ABB RobotStudio station: Project1_3.rspag

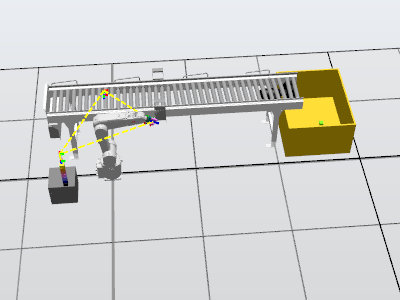
--- station ---
Station Project1 (saved by RobotStudio 23.3.10550.0)
Controller Controller1
  mechanical unit ROB_1: IRB1200_5_90_STD_03, 6 joints, base frame (0, 0, 0) mm
Layout (positions relative to the parent item):
  - My_Gripper_Mech [mechanism] at (461.39, 0, 883.1) mm, rotated rx 180 ry 60 rz 180 deg; joint values [0, 0] (rad or m)
      TCP My_Gripper_Mech_1 at (0, 0, 70) mm
      links: L1, L2, L3
  - LineSensor [smart component, from Components\LineSensor.rslib] at (522.01, 0, 848.1) mm, rotated rx 180 ry 60 rz 180 deg
      properties: Start=[0 0 0]; End=[0 0 0.1]; Length=0.1; Radius=0; Tag=(none); SensedPart=(none); SensedPoint=[0 0 0]
    - _sensorPart_ [part, from Components\LineSensor.rslib]
  - Attacher [smart component, from Components\Attacher.rslib]
      properties: Parent=IRB1200_5_90_STD_03; Flange=0; Child=(none); Mount=false; Offset=[0 0 0]; Orientation=[0 0 0]
  - Detacher [smart component, from Components\Detacher.rslib]
      properties: Child=(none); KeepPosition=true
  - PoseMover [smart component, from Components\PoseMover.rslib]
      properties: Mechanism=My_Gripper_Mech; Pose=1; Duration=0
  - PoseMover_2 [smart component, from Components\PoseMover.rslib]
      properties: Mechanism=My_Gripper_Mech; Pose=2; Duration=0
  - puelko [part] at (-800, -100, 0) mm, size 800 x 1000 x 500 mm
  - klocek8 [part] at (-525, -400, 300) mm, size 50 x 50 x 50 mm
  - klocek7 [part] at (-525, -400, 350) mm, size 50 x 50 x 50 mm
  - klocek6 [part] at (-525, -400, 400) mm, size 50 x 50 x 50 mm
  - IRB1200_5_90_STD_03 [mechanism, from %ABB.RobotStudio.Models.IRB1200%\IRB1200_5_90_STD_03.rslib] at (0, 0, 0) mm; joint values [0, -0.1239, 0.0383, 0, 0.6093, 0] (rad or m)
  - 400_guide [part, from %ABB.RobotStudio.Models.Conveyors%\Conveyor Guide 400.rslib] at (-700, 401, -100) mm
  - klocek3 [part] at (-525, -400, 550) mm, size 50 x 50 x 50 mm
  - klocek5 [part] at (-525, -400, 450) mm, size 50 x 50 x 50 mm
  - klocek4 [part] at (-525, -400, 500) mm, size 50 x 50 x 50 mm
  - Part_1 [part] at (0, -100, 0) mm, size 300 x 300 x 200 mm
  - klocek2 [part] at (-525, -400, 600) mm, size 50 x 50 x 50 mm
  - klocek1 [part] at (2609.57, 581.28, -0.23) mm, rotated rx -89.6 ry -89.83 rz -4.57 deg, size 50 x 50 x 50 mm
  - Part_3 [part] at (0, 0, 0) mm, size 300 x 300 x 100 mm
Attachment: LineSensor is attached to My_Gripper_Mech / L1
Attachment: My_Gripper_Mech is attached to IRB1200_5_90_STD_03 / Link6
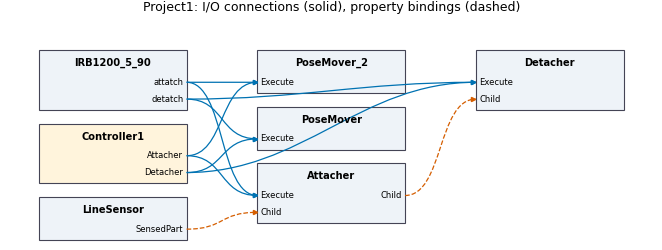
Station logic (signal -> signal, property => property):
  IRB1200_5_90.attatch -> Attacher.Execute
  IRB1200_5_90.detatch -> Detacher.Execute
  IRB1200_5_90.attatch -> PoseMover_2.Execute
  IRB1200_5_90.detatch -> PoseMover.Execute
  Controller1.Attacher -> Attacher.Execute
  Controller1.Detacher -> Detacher.Execute
  Controller1.Attacher -> PoseMover_2.Execute
  Controller1.Detacher -> PoseMover.Execute
  Attacher.Child => Detacher.Child
  LineSensor.SensedPart => Attacher.Child

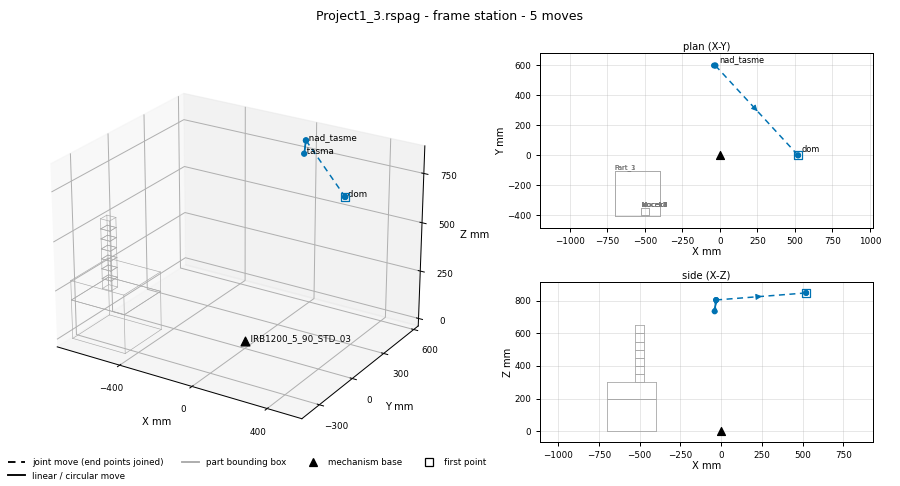
[picture p0: tool path of Project1_3.rspag in frame station, 5 of 8 moves have a stored position in this frame; points joined in program order, loops and branches not executed]
--- Controller Data/Controller1/RAPID/TASK1/PROGMOD/CalibData.mod ---
MODULE CalibData
    PERS tooldata My_Gripper_Mech_1:=[TRUE,[[0,0,70],[1,0,0,0]],[1,[1,1,1],[1,0,0,0],0,0,0]];
    TASK PERS wobjdata Workobject_1:=[FALSE,TRUE,"",[[0,0,0],[1,0,0,0]],[[0,0,0],[1,0,0,0]]];
    PERS tooldata My_Gripper_Mech_1_2:=[TRUE,[[0,0,70],[1,0,0,0]],[1,[1,1,1],[1,0,0,0],0,0,0]];
ENDMODULE

--- Controller Data/Controller1/RAPID/TASK1/PROGMOD/Module1.mod ---
MODULE Module1
    CONST robtarget dom:=[[522.01408311,0,848.1],[0.5,0,0.866025404,0],[0,0,0,0],[9E+09,9E+09,9E+09,9E+09,9E+09,9E+09]];
    CONST robtarget nad_klocek:=[[-500,-375,810],[0,0.707106781,0.707106781,0],[-2,0,-1,0],[9E+09,9E+09,9E+09,9E+09,9E+09,9E+09]];
    CONST robtarget klocek:=[[-500,-375,700],[0,0.707106781,0.707106781,0],[-2,0,-1,0],[9E+09,9E+09,9E+09,9E+09,9E+09,9E+09]];
    CONST robtarget nad_tasme:=[[-30.156,599.226,805],[0,1,0,0],[0,0,-2,0],[9E+09,9E+09,9E+09,9E+09,9E+09,9E+09]];
    CONST robtarget tasma:=[[-39.156,599.226,735],[0,1,0,0],[0,0,-2,0],[9E+09,9E+09,9E+09,9E+09,9E+09,9E+09]];
    VAR robtarget nad_klocekvar;
    VAR robtarget klocekvar;
    PROC Path_10()
        FOR z FROM 0 TO 0 DO
            nad_klocekvar:=Offs(nad_klocek,0,0,z*(-50));
            klocekvar:=Offs(klocek,0,0,z*(-50));
            tower;
        ENDFOR
        WaitTime 5;
    ENDPROC
    PROC tower()
        MoveL dom,v1000,z100,My_Gripper_Mech_1\WObj:=Workobject_1;
        SetDO Attacher,0;
        SetDO Detacher,1;
        MoveJ nad_klocekvar,v1000,z100,My_Gripper_Mech_1\WObj:=Workobject_1;
        WaitTime 0.5;
        MoveL klocekvar,v1000,z100,My_Gripper_Mech_1\WObj:=Workobject_1;
        SetDO Detacher,0;
        WaitTime 0.5;
        SetDO Attacher,1;
        WaitTime 0.3;
        MoveL nad_klocekvar,v1000,z100,My_Gripper_Mech_1\WObj:=Workobject_1;
        MoveJ nad_tasme,v1000,z100,My_Gripper_Mech_1\WObj:=Workobject_1;
        WaitTime 0.3;
        MoveL tasma,v1000,z100,My_Gripper_Mech_1\WObj:=Workobject_1;
        WaitTime 0.3;
        SetDO Detacher,1;
        SetDO Attacher,0;
        MoveL nad_tasme,v1000,z100,My_Gripper_Mech_1\WObj:=Workobject_1;
        MoveJ dom,v1000,z100,My_Gripper_Mech_1\WObj:=Workobject_1;
        WaitTime 0.1;

    ENDPROC

ENDMODULE

--- Controller Data/Controller1/SYSPAR/EIO.cfg ---
EIO:CFG_1.0:6:1::
#
EIO_SIGNAL:

      -Name "D10_2" -SignalType "DO" -Access "All"

      -Name "Attacher" -SignalType "DO" -Access "All"

      -Name "Detacher" -SignalType "DO" -Access "All"
